SUBAPPLICATION Uebung_110 (* Übung zum Integer Überlauf *)
  (* Standard: 61499-2; Description: Copyright (c) 2023 Meisterschulen am Ostbahnhof This program and the accompanying materials are made available under the terms of the Eclipse Public License 2.0 which is available at https://www.eclipse.org/legal/epl-2.0/ SPDX-License-Identifier: EPL-2.0 *)
  (* Version 1.0, 2023-10-23, Franz Höpfinger, Meisterschulen am Ostbahnhof *)
  PACKAGE Uebungen;
  IMPORT logiBUS::io::DI::logiBUS_DI::Input_I1;
  IMPORT logiBUS::io::DI::logiBUS_DI_Events::BUTTON_SINGLE_CLICK;
  IMPORT logiBUS::io::DQ::logiBUS_DO::Output_Q1;
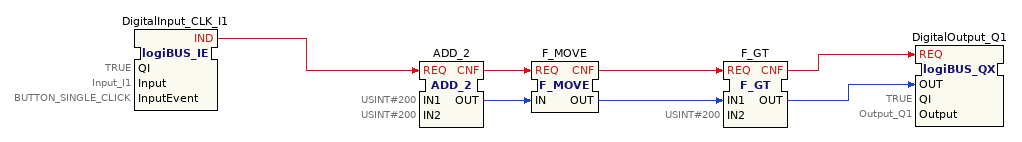
  (* Arithmetischer Überlauf https://de.wikipedia.org/wiki/Arithmetischer_%C3%9Cberlauf https://www.youtube.com/watch?v=TLanGc-c9Ww *)
  FBS
    DigitalOutput_Q1 : logiBUS::io::DQ::logiBUS_QX(QI := TRUE, Output := Output_Q1);
    ADD_2 : iec61131::arithmetic::ADD_2(IN1 := USINT#200, IN2 := USINT#200);
    DigitalInput_CLK_I1 : logiBUS::io::DI::logiBUS_IE(QI := TRUE, Input := Input_I1, InputEvent := BUTTON_SINGLE_CLICK);
    F_GT : iec61131::comparison::F_GT(IN2 := USINT#200);
    F_MOVE : iec61131::selection::F_MOVE; {SET_ATTRIBUTE(DataType, USINT)}
  END_FBS
  EVENT_CONNECTIONS
    DigitalInput_CLK_I1.IND TO ADD_2.REQ;
    F_MOVE.CNF TO F_GT.REQ;
    F_GT.CNF TO DigitalOutput_Q1.REQ;
    ADD_2.CNF TO F_MOVE.REQ;
  END_CONNECTIONS
  DATA_CONNECTIONS
    F_MOVE.OUT TO F_GT.IN1;
    F_GT.OUT TO DigitalOutput_Q1.OUT;
    ADD_2.OUT TO F_MOVE.IN;
  END_CONNECTIONS
END_SUBAPPLICATION
